PROGRAM MAIN
VAR
	fbBandMotor : FB_Motor;
	fbOfenMotor : FB_Motor;
	
	bBandStart : BOOL;
	bBandStop : BOOL;
	bBandErr : BOOL;
	bBandReset : BOOL;
	
	bOfenStart : BOOL;
	bOfenStop : BOOL;
	bOfenErr : BOOL;
	bOfenReset : BOOL;
END_VAR

fbBandMotor(
	bStart := bBandStart,
	bStop := bBandStop,
	bThermalErr := bBandErr,
	bReset := bBandReset
);

fbOfenMotor(
	bStart := bOfenStart,
	bStop := bOfenStop,
	bThermalErr := bOfenErr,
	bReset := bOfenReset
);

END_PROGRAM

(* stored: Version 1.1.0.1
   POU MAIN: Id {91985950-1f0c-4719-8dd8-725f5508eb01}, SpecialFunc None *)
